TYPE Offeset_Apprendimento :
STRUCT
	Lastra 	: StrutturaGenericaQuotaAssi;
	Falda 	: StrutturaGenericaQuotaAssi;
END_STRUCT
END_TYPE

(* stored: Version 1.1.0.1, ProductVersion 3.1.4024.11
   DUT Offeset_Apprendimento: Id {6ffd58cf-656b-4441-aefe-fc72bd82ed59} *)
